Fanuc KAREL source: kb00143.KL

-- PROVISIONAL review KL for V940-1; original PC SHA256 5a07ac9824b6da06c050a21075476e37a40544ae636a9b1f863692a810411fc3
-- Incomplete behavior may be omitted. Consult companion uncertainty JSON. Do not deploy.
PROGRAM KB00143
%NOLOCKGROUP
BEGIN
  -- V9_ZERO_TABLE_METADATA_HINT layout=0002_ascii; no indexed target words; source/name/runtime held
  -- UNRESOLVED_PC offsets 5-14; opcodes 3F,75
  -- UNRESOLVED_PC offsets 19-26; opcodes 9D,23
  -- UNRESOLVED_PC offsets 31-38; opcodes 9D,23
  -- UNRESOLVED_PC offsets 43-73; opcodes 27,22,2A,22,22,22,31
  -- UNRESOLVED_PC offsets 78-82; opcodes 7F
END KB00143
